(* CODESYS project AuroTextile_PrintingMC_04_03_20.project
   Title: AuroTextile_PrintingMC
   Version: 0.0.0.0

Project tree, tasks and I/O mapping:
  MyController : TM218LDAE24DRHN, Schneider Electric, order no. TM218LDAE24DRHN, version 4.0.1.26
      settings: Expansion Tasks.Expansion 1 Task Name = 'MAST'
    application Application
      libraries: Standard, * (System); FloatingToReal, 0.0.0.1 (SublimeAutomation); CAA File, 3.5.3.132 (CAA Technical Workgroup); SysTimeRtc, 3.5.1.0 (System)
      task MAST (cyclic, interval 100 ms, priority 15, watchdog t#1s x 1) calls MyPOU, RPi_Reporting
      task MAST_Total (cyclic, interval t#500ms, priority 1, watchdog t#1s x 1) calls TotalFlow
      function HiddenPOU [ST]
      global variables GVL
      program MyPOU [FBD]
      program TotalFlow [FBD]
      global variables GVL_RPi
      program RPi_Reporting [ST]
      function block averageReal [ST]
    Embedded Functions
      IO : IO, Schneider Electric, version 4.0.1.26
          input  iwIO_IW0 : WORD  // IW0
          input  iStart : BOOL  // IW0.I4
          input  iStop : BOOL  // IW0.I5
          input  iReset : BOOL  // IW0.I6
          input  iPower : BOOL  // IW0.I7
          output qStartIL : BOOL  // QW0.Q0
          unmapped channels: QW0
      HSC : HSC, Schneider Electric, version 4.0.1.26
          settings: HSC00VarName = 'HSC00'; HSC02VarName = 'HSC02'
    Serial Line 1
      Modbus_Manager_1 : Modbus Manager, Schneider Electric, version 4.0.0.2
    Serial Line 2
      Modbus_Manager : Modbus Manager, Schneider Electric, version 4.0.0.2
    Ethernet
        settings: IPAddress = [192, 168, 1, 10]; SubnetMask = [255, 255, 255, 0]; WebServer = FALSE; FTP Server = FALSE; SoMachine Protocol = TRUE; Modbus Server = TRUE; NetManage Protocol = FALSE; SNMP protocol = FALSE; Enable Routing = FALSE
    Module_1 : TM2AMI4HTN, Schneider Electric, order no. TM2AMI4HTN, version 4.0.1.26
        settings: IW0.Maximum = 15000; IW2.Maximum = 28000
        input  iwAirMeter : INT  // IW0
        input  iwWaterMeter : INT  // IW2
        unmapped channels: IW1, IW3
*)

// MyController/Application/GVL
VAR_GLOBAL
	hsc1error: BOOL;
	hsc1RunFB: BOOL;
	hsc1ModuloFlag: BOOL;
	hsc1ResetModulo: BOOL;
	resetLength: BOOL;
	hsc2error: BOOL;
	hsc2RunFB: BOOL;
	
	finalLength AT %MD5: REAL;
	kWhReading AT %MD6: REAL;
	kVAhReading AT %MD7: REAL;
	kWReading AT %MD8: REAL;
	thermicFlowReal AT %MD9: REAL;
	thermicTotalReal AT %MD10: REAL;
	waterFlow AT %MD11: REAL;
	waterTotal AT %MD12: REAL;
	airFlow AT %MD13: REAL;
	airTotal AT %MD14: REAL;
	speedMeasured AT %MD15: REAL;
	
	powerStatus: INT;
	currYear : INT;
	currMonth	: INT;
	currDay : INT;
	currHour : INT;
	currMinute : INT;
	currSeconds : INT;
	
	//lengthFloat: FLOAT;
	currDTString: STRING[20];
END_VAR

VAR_GLOBAL RETAIN
	CTU_0: CTU;
	moduloCountWord: WORD;
	lengthMeasured: REAL;
	lengthSaved: REAL;
	hsc1CurrVal: DINT;
	hsc2CurrVal: DINT;
	shaftDiameter  AT %MD30: REAL := 170;
	encoderPPR AT %MD31: REAL := 1024;
	productCode AT %MB0: STRING[12]; //at %MW0 to %MW6. 12 characters. One byte for each character and One extra byte.
	runStatus AT %MW100: INT;
	stopCode AT %MW101: INT;
	productType AT %MW102: INT;
	startDisabled AT %MX400.0 : BOOL;
	selectMulti AT %MX400.1 : BOOL;
	stopDTString AT %MB2600: STRING[20];
	stopCode2 AT %MW1312: INT;
END_VAR

// MyController/Application/GVL_RPi
VAR_GLOBAL
	productCode_RPi AT %MB2000: STRING[12]; //at %MW0 to %MW6. 12 characters. One byte for each character and One extra byte.
	productType_RPi AT %MW1007: INT;
	runStatus_RPi AT %MW1008: INT;
	powerStatus_RPi AT %MW1009: INT;
	stopCode_RPi AT %MW1010: INT;
	speed_RPi AT %MW1011: UINT;
	finalLength_RPi AT %MW1012: INT;
	lengthExp AT %MW1013: INT;
	airFlow_RPi AT %MW1014: INT;
	airExp AT %MW1015: INT;
	airTotal_RPi AT %MW1016: INT;
	airTotExp AT %MW1017: INT;
	waterFlow_RPi AT %MW1018: INT;
	waterExp AT %MW1019: INT;
	waterTotal_RPi AT %MW1020: INT;
	waterTotExp AT %MW1021: INT;
	thermicFlow_RPi AT %MW1022: INT;
	thermicExp AT %MW1023: INT;
	thermicTotal_RPi AT %MW1024: INT;
	thermicTotExp AT %MW1025: INT;
	kWReading_RPi AT %MW1026: INT;
	kwExp AT %MW1027: INT;
	kWhReading_RPi AT %MW1028: INT;
	kWhExp AT %MW1029: INT;
	kVAhReading_RPi AT %MD516: DINT;
	
	
END_VAR

// MyController/Application/MyPOU
PROGRAM MyPOU
VAR	
	R_TRIG_0: R_TRIG;
	TON_0: TON;
	READ_VAR_0: READ_VAR;
	ADDM_0: ADDM;
	thermicFlow: ADDRESS;
	BLINK_0: BLINK;
	buff0: ARRAY[0..3] OF WORD;
	
	FloatingToReal_0: FloatingToReal;
	FloatingToReal_1: FloatingToReal;
	
	READ_VAR_1: READ_VAR;
	ADDM_1: ADDM;
	meter2Address: ADDRESS;
	meter2Buff: ARRAY[0..1] OF WORD;
	meter2Data1: WORD;
	meter2Data2: WORD;	
	meter2Busy: BOOL;
	meter1Busy: BOOL;
	meter2KVA: REAL;
	FloatingToReal_2: FloatingToReal;
	READ_VAR_2: READ_VAR;
	energyBuff: ARRAY[0..3] OF WORD;
	energyBusy: BOOL;
	kwhData1: WORD;
	kwhData2: WORD;
	kvahData1: WORD;
	kvahData2: WORD;
	FloatingToReal_3: FloatingToReal;
	FloatingToReal_4: FloatingToReal;
	get_time_result: UDINT;
	ctrl_date_time: SYSTIMEDATE;
	utc_to_date_diag: UDINT;
	F_TRIG_0: F_TRIG;
	F_TRIG_1: F_TRIG;
	averageReal_0: averageReal;
	speedActual: REAL;
	BLINK_1: BLINK;
	averageReal_1: averageReal;
	speedAvg: REAL;
END_VAR
VAR // added by the converter: edge detectors and wires of the graphical bodies
    _w1 : BOOL;
END_VAR

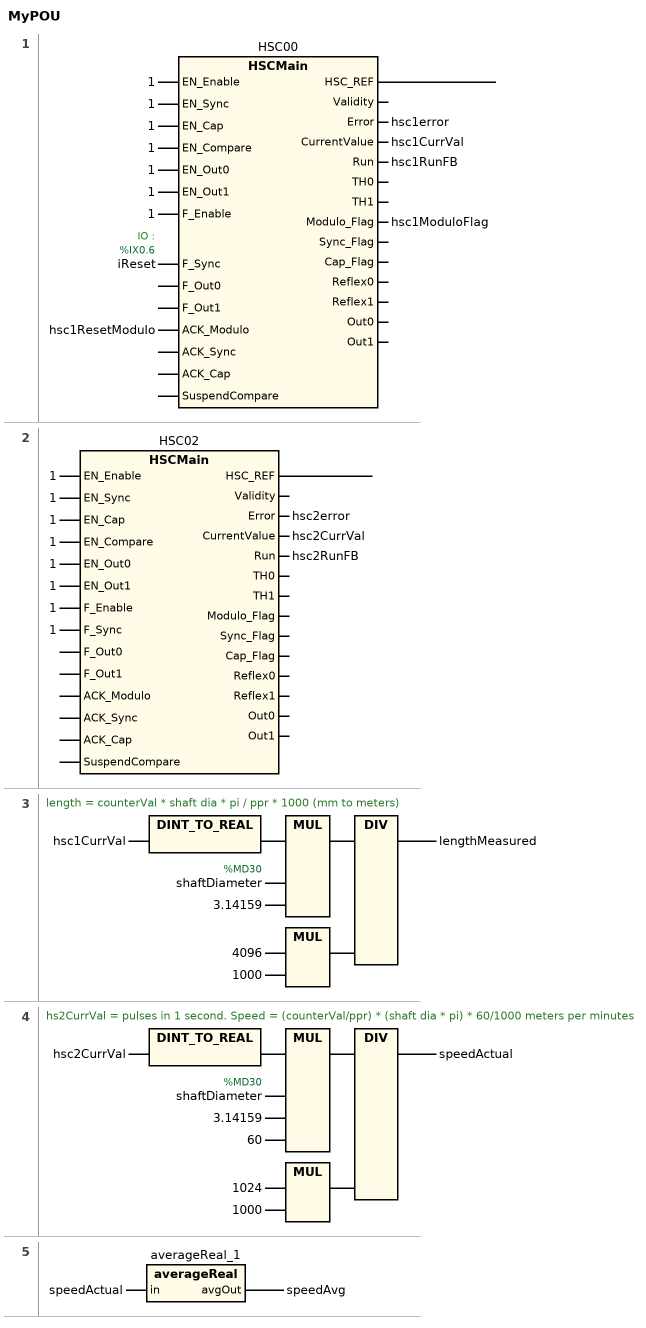
// NETWORK 1
//   iReset: IO : | AT %IX0.6
HSC00(
    EN_Enable := 1,
    EN_Sync := 1,
    EN_Cap := 1,
    EN_Compare := 1,
    EN_Out0 := 1,
    EN_Out1 := 1,
    F_Enable := 1,
    F_Sync := iReset,
    ACK_Modulo := hsc1ResetModulo,
    Error => hsc1error,
    CurrentValue => hsc1CurrVal,
    Run => hsc1RunFB,
    Modulo_Flag => hsc1ModuloFlag); // HSCMain

// NETWORK 2
HSC02(
    EN_Enable := 1,
    EN_Sync := 1,
    EN_Cap := 1,
    EN_Compare := 1,
    EN_Out0 := 1,
    EN_Out1 := 1,
    F_Enable := 1,
    F_Sync := 1,
    Error => hsc2error,
    CurrentValue => hsc2CurrVal,
    Run => hsc2RunFB); // HSCMain

// NETWORK 3
// length = counterVal * shaft dia * pi / ppr * 1000 (mm to meters)
//   shaftDiameter: AT %MD30
lengthMeasured := (DINT_TO_REAL(hsc1CurrVal) * shaftDiameter * 3.14159) / (4096 * 1000);

// NETWORK 4
// hs2CurrVal = pulses in 1 second. Speed = (counterVal/ppr) * (shaft dia * pi) * 60/1000 meters per minutes
//   shaftDiameter: AT %MD30
speedActual := (DINT_TO_REAL(hsc2CurrVal) * shaftDiameter * 3.14159 * 60) / (1024 * 1000);

// NETWORK 5
averageReal_1(in := speedActual); // averageReal
speedAvg := averageReal_1.avgOut;

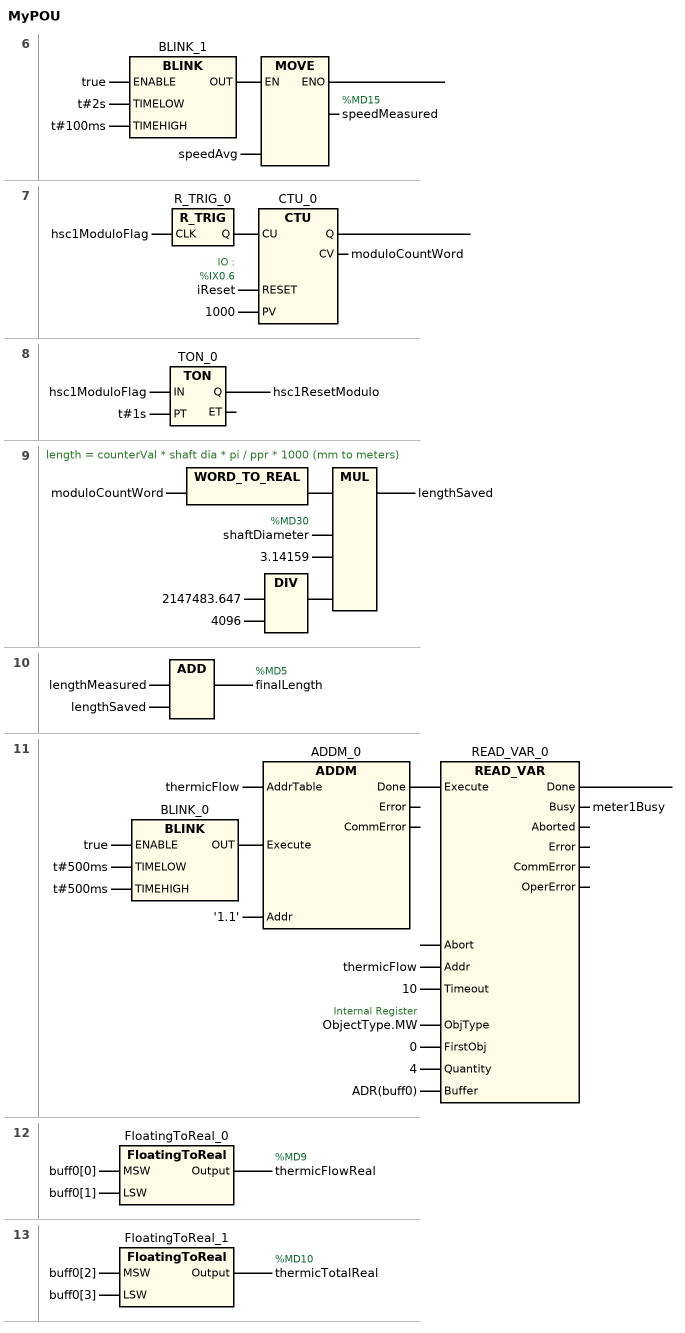
// NETWORK 6
//   speedMeasured: AT %MD15
BLINK_1(ENABLE := true, TIMELOW := t#2s, TIMEHIGH := t#100ms); // BLINK
IF BLINK_1.OUT THEN speedMeasured := speedAvg; END_IF

// NETWORK 7
//   iReset: IO : | AT %IX0.6
R_TRIG_0(CLK := hsc1ModuloFlag); // R_TRIG
CTU_0(CU := R_TRIG_0.Q, RESET := iReset, PV := 1000, CV => moduloCountWord); // CTU

// NETWORK 8
TON_0(IN := hsc1ModuloFlag, PT := t#1s); // TON
hsc1ResetModulo := TON_0.Q;

// NETWORK 9
// length = counterVal * shaft dia * pi / ppr * 1000 (mm to meters)
//   shaftDiameter: AT %MD30
lengthSaved := WORD_TO_REAL(moduloCountWord) * shaftDiameter * 3.14159 * (2147483.647 / 4096);

// NETWORK 10
//   finalLength: AT %MD5
finalLength := lengthMeasured + lengthSaved;

// NETWORK 11
//   ObjectType.MW: Internal Register
BLINK_0(ENABLE := true, TIMELOW := t#500ms, TIMEHIGH := t#500ms); // BLINK
ADDM_0(AddrTable := thermicFlow, Execute := BLINK_0.OUT, Addr := '1.1'); // ADDM
READ_VAR_0(
    Execute := ADDM_0.Done,
    Addr := thermicFlow,
    Timeout := 10,
    ObjType := ObjectType.MW,
    FirstObj := 0,
    Quantity := 4,
    Buffer := ADR(buff0),
    Busy => meter1Busy); // READ_VAR

// NETWORK 12
//   thermicFlowReal: AT %MD9
FloatingToReal_0(MSW := buff0[0], LSW := buff0[1]); // FloatingToReal
thermicFlowReal := FloatingToReal_0.Output;

// NETWORK 13
//   thermicTotalReal: AT %MD10
FloatingToReal_1(MSW := buff0[2], LSW := buff0[3]); // FloatingToReal
thermicTotalReal := FloatingToReal_1.Output;

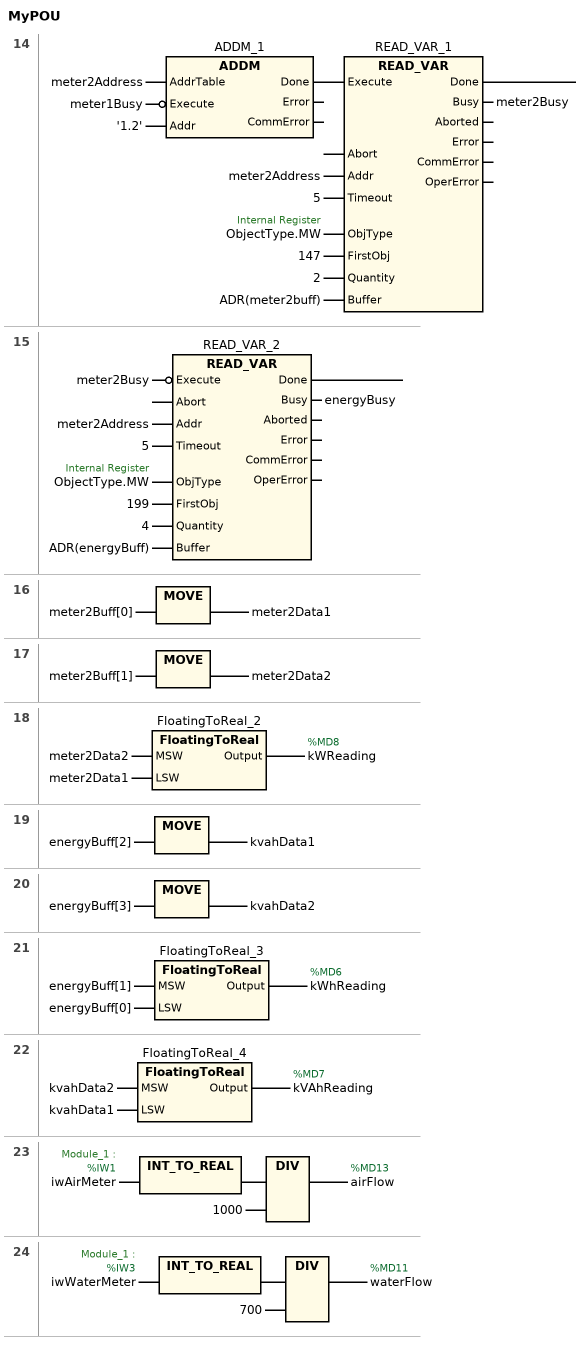
// NETWORK 14
//   ObjectType.MW: Internal Register
ADDM_1(AddrTable := meter2Address, Execute := NOT meter1Busy, Addr := '1.2'); // ADDM
READ_VAR_1(
    Execute := ADDM_1.Done,
    Addr := meter2Address,
    Timeout := 5,
    ObjType := ObjectType.MW,
    FirstObj := 147,
    Quantity := 2,
    Buffer := ADR(meter2buff),
    Busy => meter2Busy); // READ_VAR

// NETWORK 15
//   ObjectType.MW: Internal Register
READ_VAR_2(
    Execute := NOT meter2Busy,
    Addr := meter2Address,
    Timeout := 5,
    ObjType := ObjectType.MW,
    FirstObj := 199,
    Quantity := 4,
    Buffer := ADR(energyBuff),
    Busy => energyBusy); // READ_VAR

// NETWORK 16
meter2Data1 := meter2Buff[0];

// NETWORK 17
meter2Data2 := meter2Buff[1];

// NETWORK 18
//   kWReading: AT %MD8
FloatingToReal_2(MSW := meter2Data2, LSW := meter2Data1); // FloatingToReal
kWReading := FloatingToReal_2.Output;

// NETWORK 19
kvahData1 := energyBuff[2];

// NETWORK 20
kvahData2 := energyBuff[3];

// NETWORK 21
//   kWhReading: AT %MD6
FloatingToReal_3(MSW := energyBuff[1], LSW := energyBuff[0]); // FloatingToReal
kWhReading := FloatingToReal_3.Output;

// NETWORK 22
//   kVAhReading: AT %MD7
FloatingToReal_4(MSW := kvahData2, LSW := kvahData1); // FloatingToReal
kVAhReading := FloatingToReal_4.Output;

// NETWORK 23
//   iwAirMeter: Module_1 : | AT %IW1
//   airFlow: AT %MD13
airFlow := INT_TO_REAL(iwAirMeter) / 1000;

// NETWORK 24
//   iwWaterMeter: Module_1 : | AT %IW3
//   waterFlow: AT %MD11
waterFlow := INT_TO_REAL(iwWaterMeter) / 700;

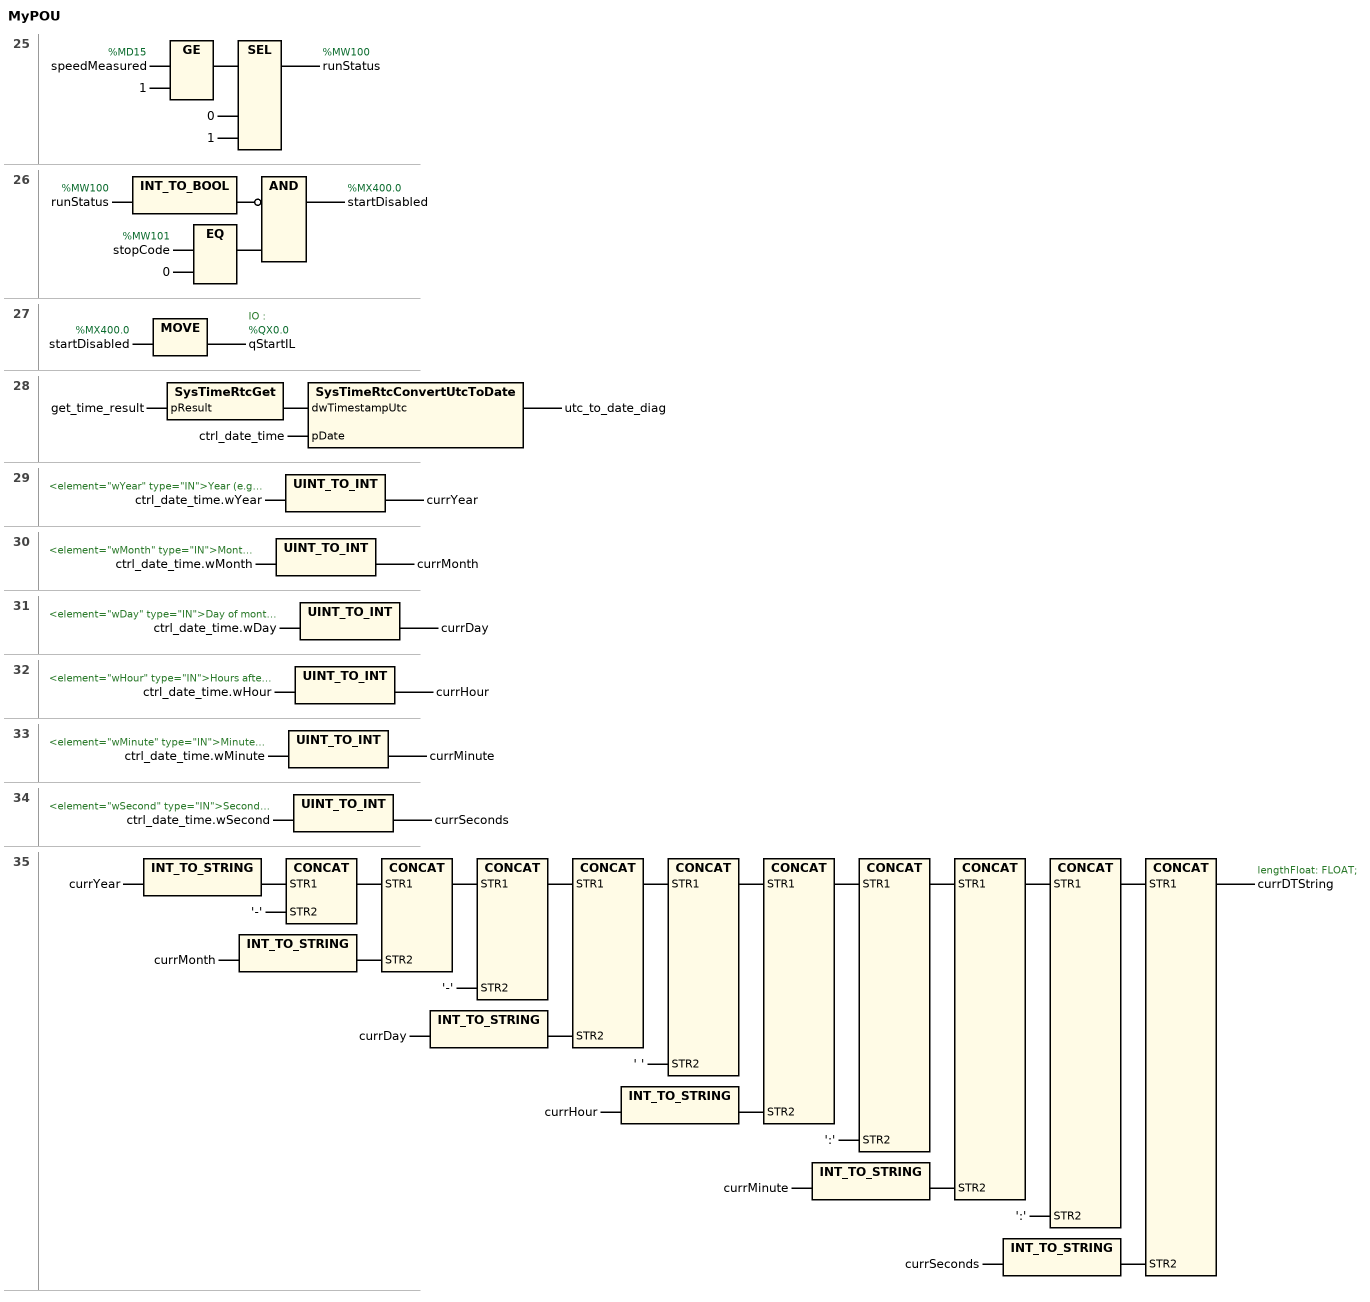
// NETWORK 25
//   speedMeasured: AT %MD15
//   runStatus: AT %MW100
runStatus := SEL(speedMeasured >= 1, 0, 1);

// NETWORK 26
//   runStatus: AT %MW100
//   stopCode: AT %MW101
//   startDisabled: AT %MX400.0
startDisabled := NOT INT_TO_BOOL(runStatus) AND stopCode = 0;

// NETWORK 27
//   startDisabled: AT %MX400.0
//   qStartIL: IO : | AT %QX0.0
qStartIL := startDisabled;

// NETWORK 28
utc_to_date_diag := SysTimeRtcConvertUtcToDate(dwTimestampUtc := SysTimeRtcGet(pResult := get_time_result), pDate := ctrl_date_time);

// NETWORK 29
//   ctrl_date_time.wYear: <element="wYear" type="IN">Year (e.g. 2006)</element>
currYear := UINT_TO_INT(ctrl_date_time.wYear);

// NETWORK 30
//   ctrl_date_time.wMonth: <element="wMonth" type="IN">Month (1..12: January = 1, December = 12)</element>
currMonth := UINT_TO_INT(ctrl_date_time.wMonth);

// NETWORK 31
//   ctrl_date_time.wDay: <element="wDay" type="IN">Day of month (1..31)</element>
currDay := UINT_TO_INT(ctrl_date_time.wDay);

// NETWORK 32
//   ctrl_date_time.wHour: <element="wHour" type="IN">Hours after midnight (0..23)</element>
currHour := UINT_TO_INT(ctrl_date_time.wHour);

// NETWORK 33
//   ctrl_date_time.wMinute: <element="wMinute" type="IN">Minutes after hour (0..59)</element>
currMinute := UINT_TO_INT(ctrl_date_time.wMinute);

// NETWORK 34
//   ctrl_date_time.wSecond: <element="wSecond" type="IN">Seconds after minute (0..59)</element>
currSeconds := UINT_TO_INT(ctrl_date_time.wSecond);

// NETWORK 35
//   currDTString: lengthFloat: FLOAT;
currDTString := CONCAT(STR1 := CONCAT(STR1 := CONCAT(STR1 := CONCAT(STR1 := CONCAT(STR1 := CONCAT(STR1 := CONCAT(STR1 := CONCAT(STR1 := CONCAT(STR1 := CONCAT(STR1 := INT_TO_STRING(currYear), STR2 := '-'), STR2 := INT_TO_STRING(currMonth)), STR2 := '-'), STR2 := INT_TO_STRING(currDay)), STR2 := ' '), STR2 := INT_TO_STRING(currHour)), STR2 := ':'), STR2 := INT_TO_STRING(currMinute)), STR2 := ':'), STR2 := INT_TO_STRING(currSeconds));

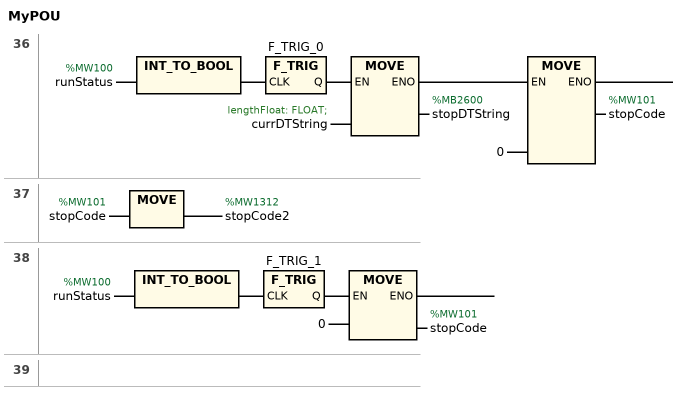
// NETWORK 36
//   runStatus: AT %MW100
//   currDTString: lengthFloat: FLOAT;
//   stopDTString: AT %MB2600
//   stopCode: AT %MW101
F_TRIG_0(CLK := INT_TO_BOOL(runStatus)); // F_TRIG
_w1 := F_TRIG_0.Q;
IF _w1 THEN stopDTString := currDTString; END_IF
IF _w1 THEN stopCode := 0; END_IF

// NETWORK 37
//   stopCode: AT %MW101
//   stopCode2: AT %MW1312
stopCode2 := stopCode;

// NETWORK 38
//   runStatus: AT %MW100
//   stopCode: AT %MW101
F_TRIG_1(CLK := INT_TO_BOOL(runStatus)); // F_TRIG
IF F_TRIG_1.Q THEN stopCode := 0; END_IF

// NETWORK 39

END_PROGRAM

// MyController/Application/averageReal
FUNCTION_BLOCK averageReal
VAR_INPUT
	in: REAL;
END_VAR
VAR_OUTPUT
	avgOut: REAL;
END_VAR
VAR
	blink_0: BLINK;
	ctu1: CTU;
	var1: REAL;
	var2: REAL;
	var3: REAL;
	var4: REAL;
	var5: REAL;
	var6: REAL;
	var7: REAL;
	var8: REAL;
	var9: REAL;
	var10: REAL;
	ctuReset: BOOL;
END_VAR

blink_0(ENABLE:=TRUE, timelow:=T#500MS, timehigh := T#50MS);
ctu1(CU:=blink_0.OUT, RESET:=ctuReset, PV:=10);

CASE ctu1.CV OF 
	1:	var1 := in;
	2:	var2 := in;
	3:	var3 := in;
	4:	var4 := in;
	5:	var5 := in;
	6:	var6 := in;
	7:	var7 := in;
	8:	var8 := in;
	9:	var9 := in;
	0:	var10 := in;
END_CASE

avgOut := (var1+var2+var3+var4+var5+var6+var7+var8+var9+var10)/10;

IF ctu1.Q THEN
	ctuReset := TRUE;
ELSE
	ctuReset := FALSE;
END_IF

END_FUNCTION_BLOCK

// MyController/Application/RPi_Reporting
PROGRAM RPi_Reporting
VAR
	length: REAL;
	
	air: REAL;
	airTot: REAL;
	water: REAL;
	waterTot: REAL;
	thermic: REAL;
	thermicTot: REAL;
	kw: REAL;
	kwh: REAL;
END_VAR

productCode_RPi	:= productCode;
productType_RPi	:= productType;
runStatus_RPi	:= runStatus;
powerStatus_RPi	:= powerStatus;
stopCode_RPi	:= stopCode;
speed_RPi		:= REAL_TO_UINT(speedMeasured*100);
length := finalLength*100;
lengthExp := REAL_TO_INT(length/32767);
finalLength_RPi := REAL_TO_INT(length - (lengthExp*32767));

air := airFlow*1000;
airExp := REAL_TO_INT(air/32767);
airFlow_RPi := REAL_TO_INT(air - (airExp*32767));

airTot:= airTotal*1000;
airTotExp := REAL_TO_INT(airTot/32767);
airTotal_RPi := REAL_TO_INT(airTot - (airTotExp*32767));

water := waterFlow*1000;
waterExp := REAL_TO_INT(water/32767);
waterFlow_RPi := REAL_TO_INT(water - (waterExp*32767));

waterTot := waterTotal*1000;
waterTotExp := REAL_TO_INT(waterTot/32767);
waterTotal_RPi := REAL_TO_INT(waterTot - (waterTotExp*32767));

thermic := thermicFlowReal*1000;
thermicExp := REAL_TO_INT(thermic/32767);
thermicFlow_RPi := REAL_TO_INT(thermic - (thermicExp*32767));

thermicTot := thermicTotalReal*1000;
thermicTotExp := REAL_TO_INT(thermicTot/32767);
thermicTotal_RPi := REAL_TO_INT(thermicTot - (thermicTotExp*32767));

kw := kWReading*1000;
kwExp := REAL_TO_INT(kw/32767);
kWReading_RPi := REAL_TO_INT(kw - (kwExp*32767));

kwh := kWhReading*1000;
kwhExp := REAL_TO_INT(kwh/32767);
kWhReading_RPi := REAL_TO_INT(kwh - (kwhExp*32767));

//finalLength_RPi	:= REAL_TO_UINT(finalLength*100);
//airFlow_RPi		:= REAL_TO_UINT(airFlow*100);
//airTotal_RPi	:= REAL_TO_UINT(airTotal*100);
//waterFlow_RPi	:= REAL_TO_UINT(waterFlow*100);
//waterTotal_RPi	:= REAL_TO_UINT(waterTotal*100);
//thermicFlow_RPi	:= REAL_TO_UINT(thermicFlowReal*100);
//thermicTotal_RPi:= REAL_TO_UINT(thermicTotalReal*100);
//kWhReading_RPi	:= REAL_TO_UINT(kWhReading*10);
//kWReading_RPi	:= REAL_TO_UINT(kWReading*100);
//kVAhReading_RPi	:= REAL_TO_UINT(kVAhReading*10);

END_PROGRAM

// MyController/Application/TotalFlow
PROGRAM TotalFlow
VAR
END_VAR

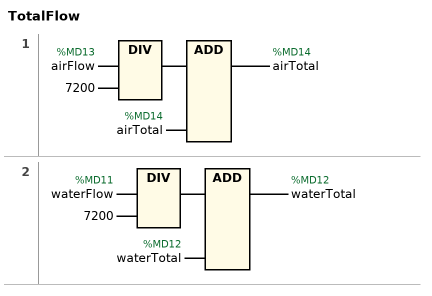
// NETWORK 1
//   airFlow: AT %MD13
//   airTotal: AT %MD14
airTotal := airFlow / 7200 + airTotal;

// NETWORK 2
//   waterFlow: AT %MD11
//   waterTotal: AT %MD12
waterTotal := waterFlow / 7200 + waterTotal;

END_PROGRAM

// MyController/Application/HiddenPOU
FUNCTION HiddenPOU : BOOL

VAR_INPUT
	pHiddenFunc: POINTER TO WORD;
END_VAR
VAR
	pRead: POINTER TO BYTE;
	pWrite: POINTER TO BYTE;
END_VAR

pRead := pHiddenFunc + 400;
pWrite := pHiddenFunc + 4400;
HiddenPOU := TRUE;

END_FUNCTION
